(* Logix 5000 project; controller Template vendor 1 type 14 code 77 rev 19.11; software revision 19.01 *)

TASK MainTask (continuous, watchdog 500 ms) : MainProgram

MODULES
   Controller : vendor 1 type 14 code 77 (CompactLogixL32EController 0, rev 19.11)
      LocalENB : 1769-L32E Ethernet Port (CompactLogixL32Ethernet 1, rev 19.11)
      Local : CompactBus (CompactVirtualAdapter 3, rev 19.11)
         Input_Module_16_PT : 1769-IQ16 (Compact 2, rev 1.1, Input RPI 2 ms)   // 16 Point Input Module Sink/Source 24VDC.
              Local:2:I.DATA.6   // Pressure_Switch
              Local:2:I.DATA.0   // Start
              Local:2:I.DATA.1   // Stop
              Local:2:I.DATA.2   // TP1
              Local:2:I.DATA.5   // TR
              Local:2:I.DATA.7   // Atmosphere
              Local:2:I   // Input
         Analog_Input_4_Chnl : 1769-IF4 (Compact 1, rev 2.1, Input RPI 2 ms)   // 4 Channel Analog Input Module.
         Output_Module_16_PT : 1769-OB16P (Compact 3, rev 2.1, Output RPI 2 ms)   // 16 Point Output Module, Fused Output.
              Local:3:O.DATA   // Output
              Local:3:O.DATA.0   // SV1
              Local:3:O.DATA.2   // SV4
              Local:3:O.DATA.3   // VV1
              Local:3:O.DATA.4   // VV2
              Local:3:O.DATA.6   // reactorheater
              Local:3:O.DATA.7   // mfcwater
END_MODULES

PROGRAM MainProgram   (* main routine MainRoutine *)
VAR
   cycles : COUNTER := (PRE := 9, ACC := 9, DN := 1);
   delay_start : TIMER := (PRE := 1000);
   done : BOOL := 1;
   done1 : BOOL := 1;
   MFC : BOOL;
   mstart : BOOL;
   mstop : BOOL := 1;
   precursor1 : INT := 1000;
   pulse_start : TIMER := (PRE := 1001);
   restart_p : TIMER;
   restart_s : TIMER := (PRE := 5);
   s_dones : BOOL;
   sdone_p : BOOL;
   section : COUNTER := (ACC := 100000000);
   start_section : TIMER := (PRE := 5000);
   start_serial : BOOL;
   startmem : BOOL;
   startpos : BOOL;
   sv11 : BOOL;
   sv1_start : BOOL;
   sv21 : BOOL;
   sv31 : BOOL;
   sv4 : BOOL;
   svac1 : BOOL;
   svac2 : BOOL;
   sw : BOOL;
   Tok : BOOL;
   tonp1 : TIMER := (PRE := 2000);
   tonp1_ons : BOOL;
   tpstart : TIMER := (PRE := 1000);
   tpvac : TIMER := (PRE := 20);
   tpvac_en : BOOL;
   trestarts : TIMER := (PRE := 1000);
   trig1 : BOOL;
   trig11 : BOOL;
   trig2 : BOOL;
   trig21 : BOOL;
   trig7 : BOOL;
   trig71 : BOOL;
   trig8 : BOOL;
   trig81 : BOOL;
   trig_tvac1 : BOOL;
   tvac1 : TIMER := (PRE := 4000);
   tvac1_start : BOOL;
   tvacw : TIMER := (PRE := 8000);
   twait1 : TIMER := (PRE := 3000);
   twaitw : TIMER := (PRE := 7000);
   twater : TIMER := (PRE := 6000);
   vacpumps : BOOL;
END_VAR

ROUTINE MainRoutine   (* ladder *)
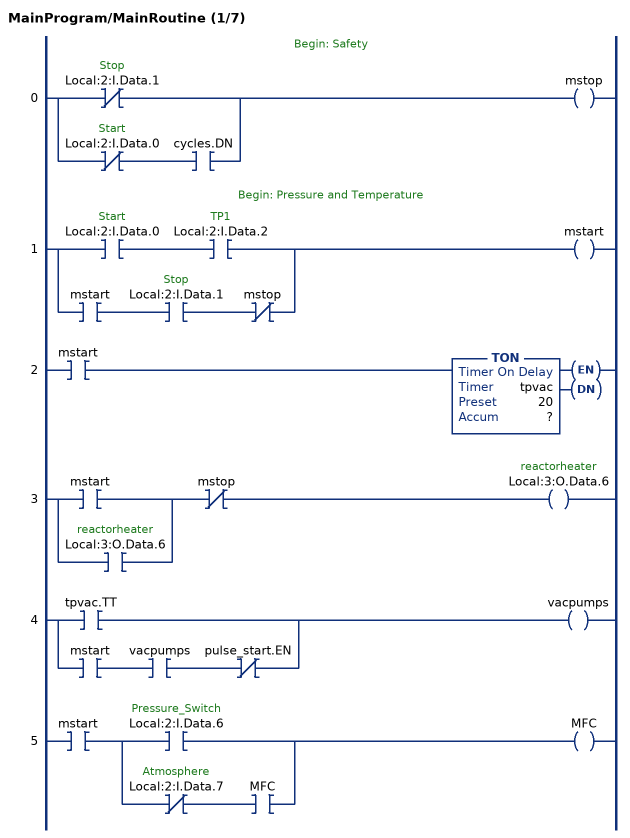
   // Begin: Safety
   0: [XIO(Local:2:I.Data.1) ,XIO(Local:2:I.Data.0) XIC(cycles.DN) ]OTE(mstop);
   // Begin: Pressure and Temperature
   1: [XIC(Local:2:I.Data.0) XIC(Local:2:I.Data.2) ,XIC(mstart) XIC(Local:2:I.Data.1) XIO(mstop) ]OTE(mstart);
   2: XIC(mstart)TON(tpvac,?,?);
   3: [XIC(mstart) ,XIC(Local:3:O.Data.6) ]XIO(mstop)OTE(Local:3:O.Data.6);
   4: [XIC(tpvac.TT) ,XIC(mstart) XIC(vacpumps) XIO(pulse_start.EN) ]OTE(vacpumps);
   5: XIC(mstart)[XIC(Local:2:I.Data.6) ,XIO(Local:2:I.Data.7) XIC(MFC) ]OTE(MFC);
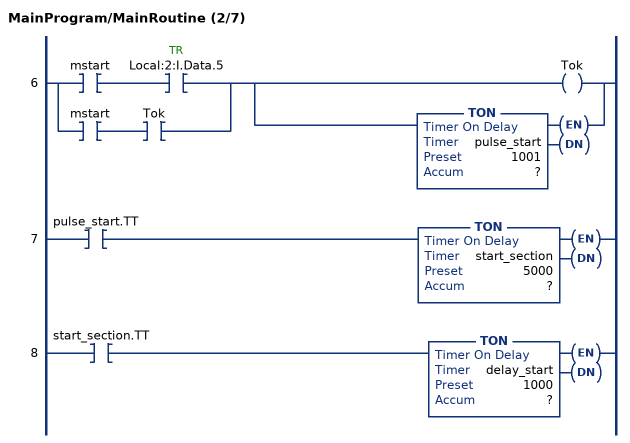
   6: [XIC(mstart) XIC(Local:2:I.Data.5) ,XIC(mstart) XIC(Tok) ][OTE(Tok) ,TON(pulse_start,?,?) ];
   7: XIC(pulse_start.TT)TON(start_section,?,?);
   8: XIC(start_section.TT)TON(delay_start,?,?);
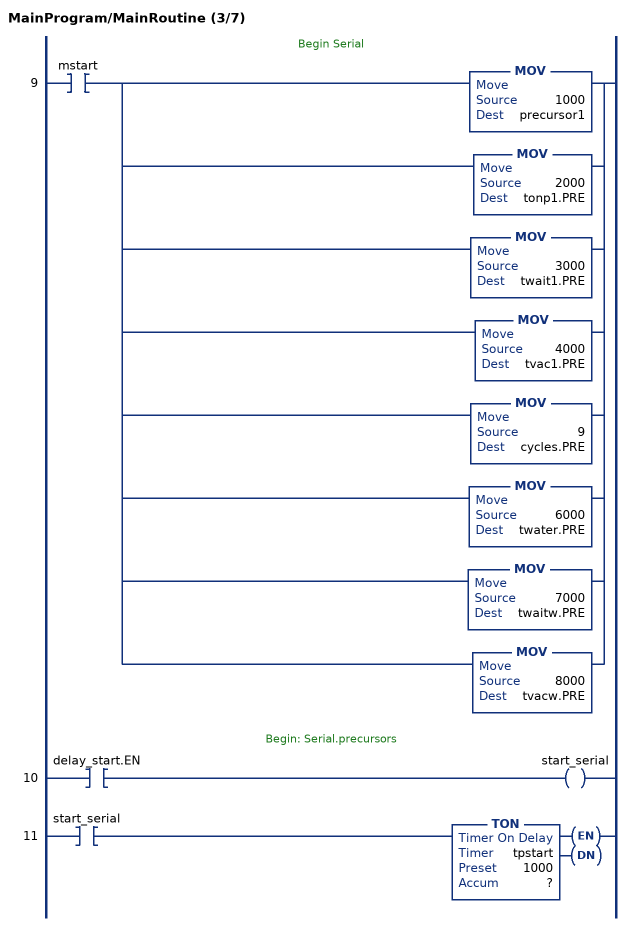
   // Begin Serial
   9: XIC(mstart)[MOV(1000,precursor1) ,MOV(2000,tonp1.PRE) ,MOV(3000,twait1.PRE) ,MOV(4000,tvac1.PRE) ,MOV(9,cycles.PRE) ,MOV(6000,twater.PRE) ,MOV(7000,twaitw.PRE) ,MOV(8000,tvacw.PRE) ];
   // Begin: Serial.precursors
   10: XIC(delay_start.EN)OTE(start_serial);
   11: XIC(start_serial)TON(tpstart,?,?);
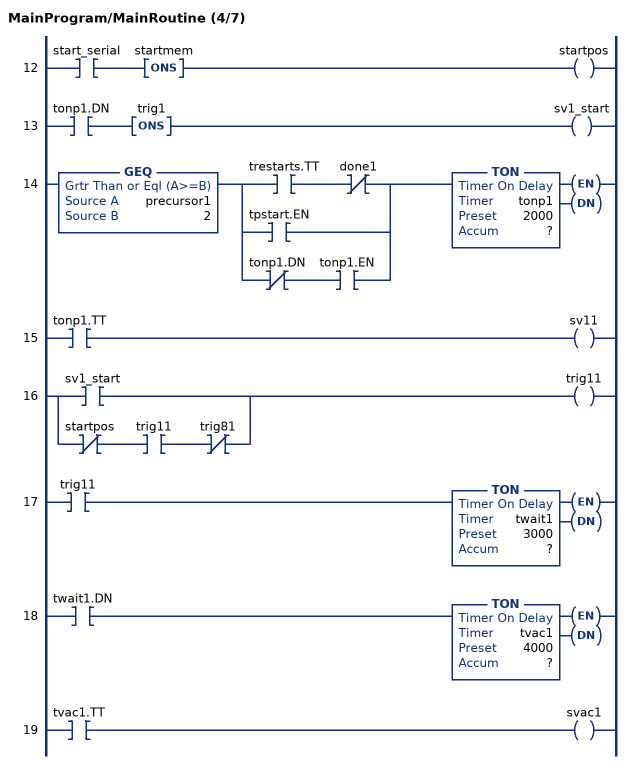
   12: XIC(start_serial)ONS(startmem)OTE(startpos);
   13: XIC(tonp1.DN)ONS(trig1)OTE(sv1_start);
   14: GEQ(precursor1,2)[XIC(trestarts.TT) XIO(done1) ,XIC(tpstart.EN) ,XIO(tonp1.DN) XIC(tonp1.EN) ]TON(tonp1,?,?);
   15: XIC(tonp1.TT)OTE(sv11);
   16: [XIC(sv1_start) ,XIO(startpos) XIC(trig11) XIO(trig81) ]OTE(trig11);
   17: XIC(trig11)TON(twait1,?,?);
   18: XIC(twait1.DN)TON(tvac1,?,?);
   19: XIC(tvac1.TT)OTE(svac1);
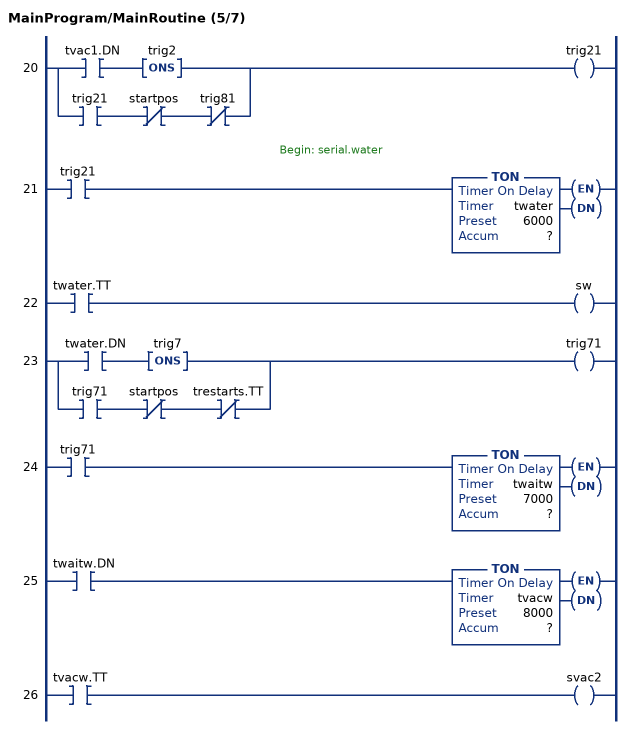
   20: [XIC(tvac1.DN) ONS(trig2) ,XIC(trig21) XIO(startpos) XIO(trig81) ]OTE(trig21);
   // Begin: serial.water
   21: XIC(trig21)TON(twater,?,?);
   22: XIC(twater.TT)OTE(sw);
   23: [XIC(twater.DN) ONS(trig7) ,XIC(trig71) XIO(startpos) XIO(trestarts.TT) ]OTE(trig71);
   24: XIC(trig71)TON(twaitw,?,?);
   25: XIC(twaitw.DN)TON(tvacw,?,?);
   26: XIC(tvacw.TT)OTE(svac2);
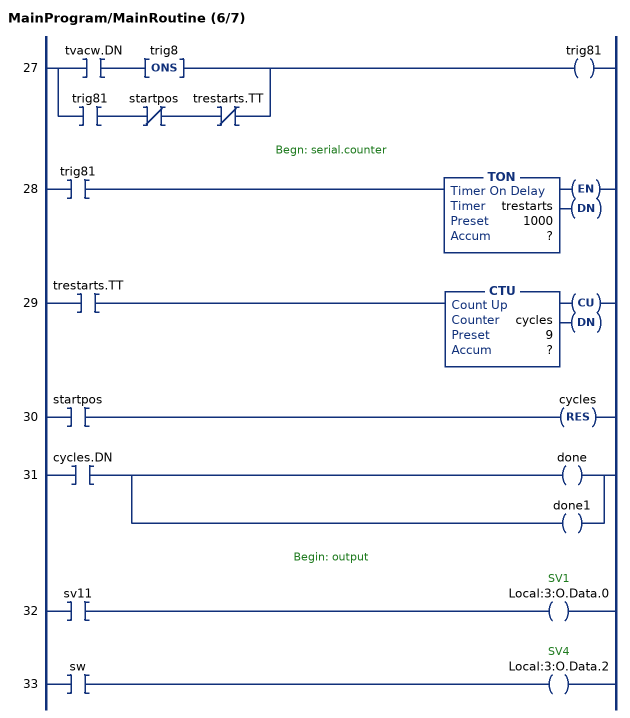
   27: [XIC(tvacw.DN) ONS(trig8) ,XIC(trig81) XIO(startpos) XIO(trestarts.TT) ]OTE(trig81);
   // Begn: serial.counter
   28: XIC(trig81)TON(trestarts,?,?);
   29: XIC(trestarts.TT)CTU(cycles,?,?);
   30: XIC(startpos)RES(cycles);
   31: XIC(cycles.DN)[OTE(done) ,OTE(done1) ];
   // Begin: output
   32: XIC(sv11)OTE(Local:3:O.Data.0);
   33: XIC(sw)OTE(Local:3:O.Data.2);
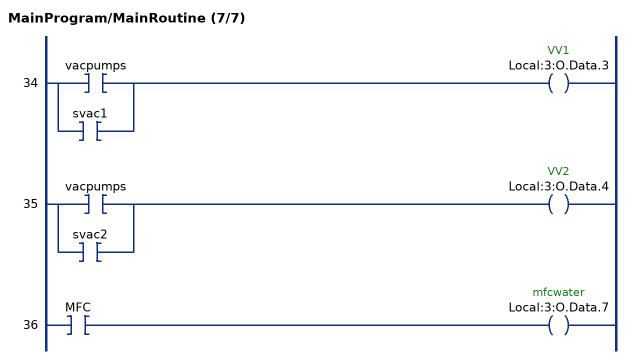
   34: [XIC(vacpumps) ,XIC(svac1) ]OTE(Local:3:O.Data.3);
   35: [XIC(vacpumps) ,XIC(svac2) ]OTE(Local:3:O.Data.4);
   36: XIC(MFC)OTE(Local:3:O.Data.7);
END_ROUTINE
END_PROGRAM

PROGRAM Template_Routine   (* main routine Template_Routine_1 *)

ROUTINE Template_Routine_1   (* ladder *)
END_ROUTINE
END_PROGRAM
